(* IEC 61131-3 sources: IRIS-Project/LASAL CONTROL SOFTWARE/LasalProject_2025_09_12/Class/ControlloServerModBus, 1 file *)

(* ---- ControlloServerModBus.st ---- *)
(*!
<Class
	Name               = "ControlloServerModBus"
	Revision           = "0.0"
	RealtimeTask       = "false"
	CyclicTask         = "true"
	DefCyclictime      = "100 ms"
	BackgroundTask     = "false"
	Sigmatek           = "false"
	OSInterface        = "false"
	HighPriority       = "false"
	Automatic          = "false"
	UpdateMode         = "Prescan"
	SharedCommandTable = "true"
	Objectsize         = "(652,120)">
	<Channels>
		<Server Name="ClassSvr" Visualized="false" Initialize="false" WriteProtected="true" Retentive="false"/>
		<Client Name="oc_ModBusTCPSlave" Required="true" Internal="false"/>
	</Channels>
</Class>
*)
ControlloServerModBus : CLASS
  //Servers:
	ClassSvr 	: SvrChCmd_DINT;
  //Clients:
	oc_ModBusTCPSlave 	: CltChCmd__ModBusTCPSLAVE;
  //Variables:
		Tempo 	: DINT;
  //Functions:

	FUNCTION VIRTUAL GLOBAL Init;

	FUNCTION VIRTUAL GLOBAL CyWork
		VAR_INPUT
			EAX 	: UDINT;
		END_VAR
		VAR_OUTPUT
			state (EAX) 	: UDINT;
		END_VAR;
  //Tables:
	FUNCTION @STD
		VAR_OUTPUT
			ret_code	: CONFSTATES;
		END_VAR;
	FUNCTION GLOBAL TAB @CT_;
END_CLASS;

#pragma usingLtd _ModBusTCPSLAVE

FUNCTION VIRTUAL GLOBAL ControlloServerModBus::CyWork
	VAR_INPUT
		EAX 	: UDINT;
	END_VAR
	VAR_OUTPUT
		state (EAX) 	: UDINT;
	END_VAR

if _FirstScan then
  oc_ModBusTCPSlave.sDisable:=1;
  oc_ModBusTCPSlave.Init();
end_if;

if oc_ModBusTCPSlave.sDisable=1 then
  Tempo:=Tempo+100;
end_if;

if Tempo=2000 then
  oc_ModBusTCPSlave.sDisable:=0;
end_if;

oc_ModBusTCPSlave.CyclicCall();

	state := READY;

END_FUNCTION

FUNCTION VIRTUAL GLOBAL ControlloServerModBus::Init

Tempo:=0;

END_FUNCTION
